TYPE E_MOTOR_RESET_STATE :
(
	MOTOR_RESET_STATE_START	:= 0,
	MOTOR_RESET_STATE_SoE_RESET,
	MOTOR_RESET_STATE_SoE_WAIT_RESET,
	MOTOR_RESET_STATE_RESET_AXIS,
	MOTOR_RESET_STATE_WAIT,
	MOTOR_RESET_STATE_END
);
END_TYPE

(* stored: Version 1.1.0.1, ProductVersion 3.1.4022.9
   DUT E_MOTOR_RESET_STATE: Id {d1f5e327-7917-4ede-a450-2022659496b6} *)
